DATA_BLOCK "LINE_3"
{ S7_Optimized_Access := 'TRUE' }
AUTHOR : RP
VERSION : 0.1
NON_RETAIN
"LINE"

BEGIN

END_DATA_BLOCK
